TYPE StructureWithStructureWithArray :
STRUCT
	myStruct : StructureWithArray;
END_STRUCT
END_TYPE

(* stored: Version 1.1.0.1, ProductVersion 3.1.4024.11
   DUT StructureWithStructureWithArray: Id {3f20319c-3773-4ad4-9341-47612ec22aa4} *)
